PROGRAM MAIN
VAR
	bBotao : BOOL;
	bHabilitado : BOOL;
END_VAR

IF bBotao THEN
	bHabilitado := TRUE;
ELSE
	bHabilitado := FALSE;
END_IF

END_PROGRAM

(* stored: Version 1.1.0.1, ProductVersion 3.1.4024.13
   POU MAIN: Id {3860ccaf-a48a-4968-aba8-5b5d2f94f2a3}, SpecialFunc None *)
